FUNCTION_BLOCK E_4States_11Transitions (* Basic FB with empty ECC *)
  (* Standard: 61499-2 *)
  (* Version 1.0, 2023-09-22, AK124910 *)
  PACKAGE servSeq;
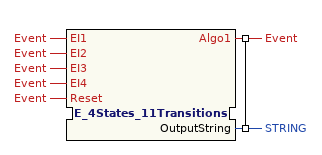
  EVENT_INPUT
    EI1;
    EI2;
    EI3;
    EI4;
    Reset;
  END_EVENT
  EVENT_OUTPUT
    Algo1 WITH OutputString;
  END_EVENT
  VAR_OUTPUT
    OutputString : STRING;
  END_VAR
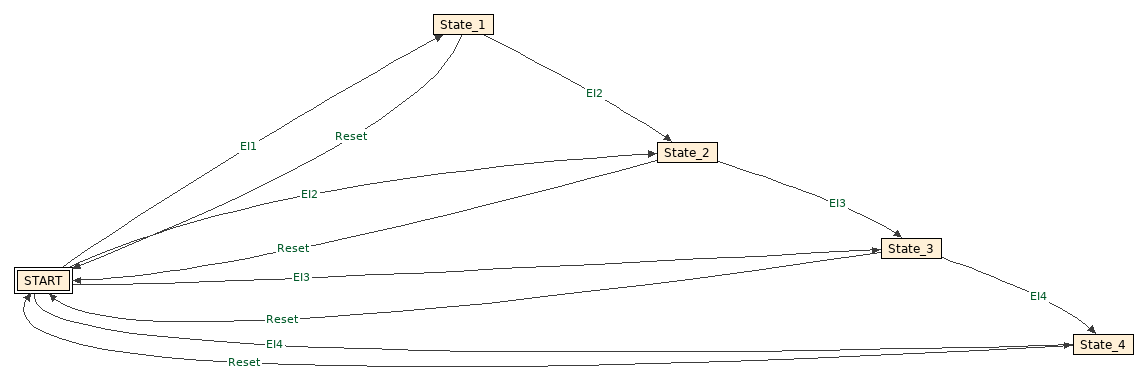
  EC_STATES
    START; (* Initial State *)
    State_1;
    State_2;
    State_3;
    State_4;
  END_STATES
  EC_TRANSITIONS
    START TO State_1 := EI1;
    State_1 TO START := Reset;
    START TO State_2 := EI2;
    State_2 TO START := Reset;
    START TO State_3 := EI3;
    State_3 TO START := Reset;
    START TO State_4 := EI4;
    State_4 TO START := Reset;
    State_1 TO State_2 := EI2;
    State_2 TO State_3 := EI3;
    State_3 TO State_4 := EI4;
  END_TRANSITIONS
  ALGORITHM HWAlgo IN ST:
OutputString := CONCAT(OutputString, 'H');
OutputString := CONCAT(OutputString, 'E');
OutputString := CONCAT(OutputString, 'L');
OutputString := CONCAT(OutputString, 'L');
OutputString := CONCAT(OutputString, 'O');
OutputString := CONCAT(OutputString, ' ');
OutputString := CONCAT(OutputString, 'W');
OutputString := CONCAT(OutputString, 'O');
OutputString := CONCAT(OutputString, 'R');
OutputString := CONCAT(OutputString, 'L');
OutputString := CONCAT(OutputString, 'D');
OutputString := CONCAT(OutputString, '!');
  END_ALGORITHM
  (* Service external/internal_interface: Basic FB with empty ECC *)
END_FUNCTION_BLOCK
